(* CODESYS project task5-1.project
   Title: Adsız
   Version: 0.0.0.0
   Author: USER

Project tree, tasks and I/O mapping:
  MyController : TM238LFDC24DT, Schneider Electric, order no. TM238LFDC24DT, version 4.0.1.28
      settings: OpcUa Enable = False
    application Application
      task MAST (cyclic, interval 20 ms, priority 15, watchdog 100 ms x 1) calls POU
      global variables GVL
      program POU [CFC]
    Embedded Functions
      IO : IO, Schneider Electric, version 4.0.1.28
          input  sensor : BOOL  // IW0.I0
          input  rst : BOOL  // IW0.I1
          output out : BOOL  // QW0.Q1
          unmapped channels: IW0, QW0
      HSC : HSC, Schneider Electric, version 4.0.1.28
      PTO_PWM : PTO_PWM, Schneider Electric, version 4.0.1.28
    Serial Line 1
      Modbus_Manager : Modbus Manager, Schneider Electric, version 4.0.0.2
    Serial Line 2
      SoMachine_Network_Manager : SoMachine-Network Manager, Schneider Electric, version 4.0.0.2
    CAN
  FdtConnections : FDT Bağlantıları, Schneider Electric, version 1.0.0.2
    Modbus_Serial_Line_Manager : Modbus Serial Line Manager, Schneider Electric, version 2.2.5
*)

// MyController/Application/GVL
VAR_GLOBAL
END_VAR

// MyController/Application/POU
PROGRAM POU
VAR
	ct: CTU;
	sdCTU_0: CTU;
	timer: TON;
END_VAR

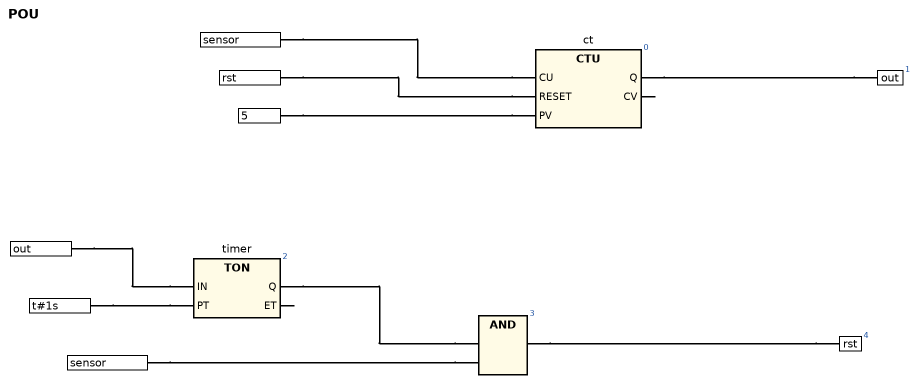
ct(CU := sensor, RESET := rst, PV := 5); // CTU
out := ct.Q;
timer(IN := out, PT := t#1s); // TON
rst := timer.Q AND sensor;

END_PROGRAM
